{attribute 'linkalways'} 
{attribute 'no_explicit_call' := 'This FB is a CLASS and must be accessed using methods or properties'}
{attribute 'enable_dynamic_creation'}
FUNCTION_BLOCK FINAL EQ_UINT EXTENDS Node
VAR
	in1 : _UINT(0);
	in2 : _UINT(0);
	out : _BOOL(FALSE);
END_VAR

METHOD PUBLIC Clone : I_Node
VAR
	pNode : POINTER TO EQ_UINT;
END_VAR
pNode := __NEW(EQ_UINT);
Clone := pNode^;
END_METHOD

METHOD FB_init : BOOL
VAR_INPUT
	bInitRetains : BOOL; // if TRUE, the retain variables are initialized (warm start / cold start)
	bInCopyCode : BOOL;  // if TRUE, the instance afterwards gets moved into the copy code (online change)
END_VAR
AddInput('in1',THIS^.in1);
AddInput('in2',THIS^.in2);
AddOutput('out', THIS^.out);
END_METHOD

METHOD PROTECTED OnExecute
VAR
END_VAR
out.Value := in1.Value = in2.Value;
END_METHOD

END_FUNCTION_BLOCK

(* stored: Version 1.1.0.1, ProductVersion 3.1.4024.15
   POU EQ_UINT: Id {763f6833-1374-4b8b-8f23-3885197907c7}, SpecialFunc None
   Folder Constructor: Id {e1099688-38c3-45ba-b931-a0dcae052eb2}
   Method Clone: Id {97b119a4-1bab-44b2-9a40-944116ced33c}
   Method FB_init: Id {1474e439-034e-4d51-b365-85ed9be59f04}
   Method OnExecute: Id {2652156e-a513-4cac-a0bf-0b1cc91d2d94} *)
